(* CoDeSys 2.3.9.62 project: Tema2Ejemplo3-CambioGiro.pro *)

(* Global variable list: Global_Variables *)
VAR_GLOBAL
  S0:BOOL;
  SI:BOOL;
  SD:BOOL;
  KM1:BOOL;
   KM2:BOOL;
END_VAR

(* POU PLC_PRG, ST *)
PROGRAM PLC_PRG
VAR
  posy:INT;
END_VAR
Control();


IF KM1=TRUE THEN
  posy:=posy-1;
END_IF

IF KM2=TRUE THEN
  posy:=posy+1;
END_IF
END_PROGRAM

(* POU Control, LD *)
PROGRAM Control
VAR
END_VAR
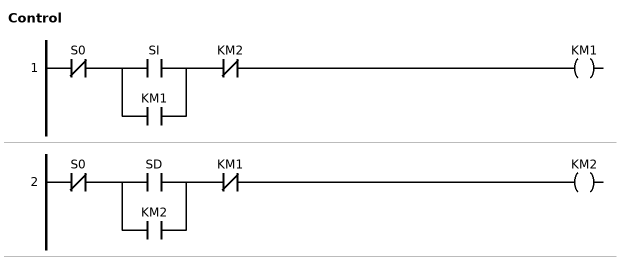
_LD_ (* Ladder Diagram *)
NETWORK 1
	[/S0] - { [SI] | [KM1] } - [/KM2] --- (KM1)
NETWORK 2
	[/S0] - { [SD] | [KM2] } - [/KM1] --- (KM2)
_END_LD_
(* the same logic as Structured Text *)
(* Network 1 *)
KM1 := NOT S0 AND (SI OR KM1) AND NOT KM2;
(* Network 2 *)
KM2 := NOT S0 AND (SD OR KM2) AND NOT KM1;
END_PROGRAM

(* Visualisation Deposito
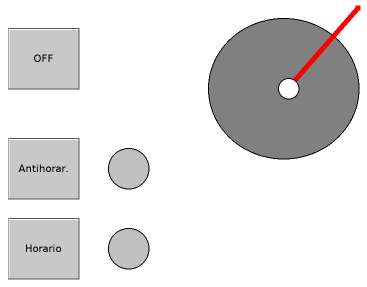
button at (50,80)-(121,141): text "OFF"; taps .S0
button at (50,190)-(121,251): text "Antihorar."; taps .SI
button at (50,270)-(121,331): text "Horario"; taps .SD
polyline at (330,60)-(400,140): angle PLC_PRG.posy
ellipse at (150,200)-(191,241): alarm colour if .KM1
ellipse at (150,280)-(191,321): alarm colour if .KM2
2 more shapes without text or variables
*)
